// TIA Portal V16 export
// export: Created 2021-11-12T13:32:28.9636488Z, ExportSetting WithDefaults, DisplayName Totally Integrated Automation Portal, DisplayVersion V16 Update 3, DisplayName TIA Portal Version Control Interface, DisplayVersion V16 Update 2, DisplayName TIA Portal Openness, DisplayVersion V16 Update 3, DisplayName SINAMICS Startdrive Advanced, DisplayVersion V16 Update 5, DisplayName SINAMICS Startdrive G130, G150, S120, S150, SINAMICS MV, S210, DisplayVersion V16 Update 5, DisplayName SINAMICS Startdrive G110M, G120, G120C, G120D, G120P, G115D, DisplayVersion V16 Update 5, DisplayName STEP 7 Professional, DisplayVersion V16 Update 3, DisplayName STEP 7 Safety, DisplayVersion V16, DisplayName WinCC UA Professional, DisplayVersion V16 Update 3
DATA_BLOCK "IDB_Station1R6"   // DB155
VERSION : 0.1
// stored: AutoNumber true, DBAccessibleFromOPCUA true, InstanceOfName Station1R6, InstanceOfType FB
"Station1R6"
   // VAR
   //    SF_RO01_Timeout : "STD_DI_Mon";
   //    "SF_CL01-BG01_Alarm" { S7_SetPoint := 'True'} : "STD_DI_Mon";
   //    "SF_CL01-BG02_Alarm" { S7_SetPoint := 'True'} : "STD_DI_Mon";
   //    SF_RC01 : "STD_DriveRobotABB";
   //    SF_RO01 : "STD_RobotABB";
   //    SF_RobotGripper : "STD_RobotGripper";
   //    SS_Edge { ExternalAccessible := 'False'; ExternalVisible := 'False'; ExternalWritable := 'False'} : Array[0..100] of Bool;
   // END_VAR
   // VAR RETAIN
   //    SDI_PartID : DInt;
   //    SI_PartType { S7_SetPoint := 'True'} : Int;
   // END_VAR
   // VAR
   //    SI_160RowNr : Int;
   //    SI_160LineNr : Int;
   //    SI_180RowNr : Int;
   //    SI_180LineNr : Int;
   //    SI_BSN2BeltExt : Int;
   //    SB1PosFound160 : Bool;
   //    SB1PosFound180 : Bool;
   //    SB1ReqToChangeTool : Bool;
   //    SB1ChangeToolDone : Bool;
   //    SB1CycleAutostop : Bool;
   //    SB1ServicePosReq { ExternalAccessible := 'False'; ExternalVisible := 'False'; ExternalWritable := 'False'} : Bool;
   //    SB1RobotInitialized : Bool;
   // END_VAR
BEGIN
END_DATA_BLOCK
